(* Schneider Machine Expert - Basic project Exercise-12 - Multiple Motor Connections with using Set Coil and Normal Coil using Latch & Memory, file version 2.9.0.0 *)
(* ProjectInformations: Name=New project *)

HARDWARE
  Cpu 0: TM221CE24R
  EthernetConfiguration: NetworkName=M221, IpAllocationMode=FixedAddress, IpAddress=0.0.0.0, SubnetMask=0.0.0.0
  SerialLineConfiguration: Baud=Baud19200, Parity=ParityEven, DataBits=DataBits8, StopBits=StopBits1, PhysicalMedium=PhysicalMediumRs485, SlaveId=1, Addressing=SlaveAddressing
  MastTask: UsePeriodScanMode=false, PeriodScan=100
  FastTask: Period=255
  CpuBehavior: StartingMode=StartAsPreviousState, AutoSaveRamOnEeprom=true, WatchdogPeriod=250

SYMBOLS  (address, symbol, comment, settings)
  %M0       MEMORY_1
  %M1       MEMORY_2
  %I0.0     SWITCH_1
  %I0.1     SWITCH_2
  %Q0.0     MOTOR_1
  %Q0.1     MOTOR_2
  %Q0.2     MOTOR_3
  %Q0.3     MOTOR_4

POU New POU
  (* SectionNumber=1 *)

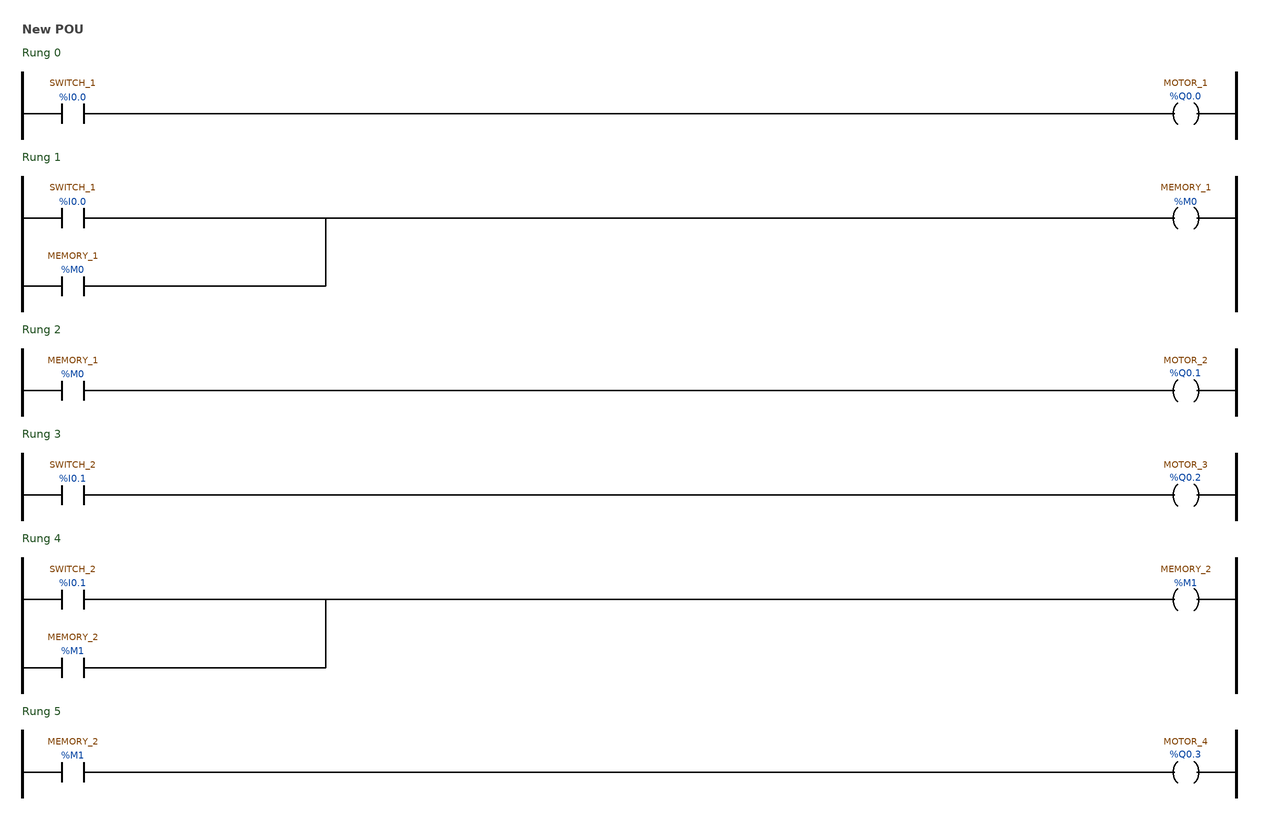

// Rung 0
  LD %I0.0                (* SWITCH_1 *)
  ST %Q0.0                (* MOTOR_1 *)
  // as ST:
  //   MOTOR_1 := SWITCH_1;

// Rung 1
  LD %I0.0                (* SWITCH_1 *)
  OR %M0                  (* MEMORY_1 *)
  ST %M0                  (* MEMORY_1 *)
  // as ST:
  //   MEMORY_1 := SWITCH_1 OR MEMORY_1;

// Rung 2
  LD %M0                  (* MEMORY_1 *)
  ST %Q0.1                (* MOTOR_2 *)
  // as ST:
  //   MOTOR_2 := MEMORY_1;

// Rung 3
  LD %I0.1                (* SWITCH_2 *)
  ST %Q0.2                (* MOTOR_3 *)
  // as ST:
  //   MOTOR_3 := SWITCH_2;

// Rung 4
  LD %I0.1                (* SWITCH_2 *)
  OR %M1                  (* MEMORY_2 *)
  ST %M1                  (* MEMORY_2 *)
  // as ST:
  //   MEMORY_2 := SWITCH_2 OR MEMORY_2;

// Rung 5
  LD %M1                  (* MEMORY_2 *)
  ST %Q0.3                (* MOTOR_4 *)
  // as ST:
  //   MOTOR_4 := MEMORY_2;
